// TIA Portal V20 export
DATA_BLOCK "Config"   // DB142
// stored: MemoryReserve 100, Namespace Unit1.Em0
   VAR
      em : "LAF_typeEmConfiguration";   // Configuration of EM Parameters
      cmStacker1NgBoxDetect : "LBC_typeDigitalSignalConfiguration";
      cmStacker1NgBoxFullDetect : "LBC_typeDigitalSignalConfiguration";
      cmStacker1NgBoxLoadingUpDown : "LBC_typeTwoWayActuatorConfiguration";
      cmStacker1NgBoxUnitMoverBwdFwd : "LBC_typeTwoWayActuatorConfiguration";
      cmStacker1NgBoxClampLeftOpenClose : "LBC_typeTwoWayActuatorConfiguration";
      cmStacker1NgBoxClampRightOpenClose : "LBC_typeTwoWayActuatorConfiguration";
      cmStacker1NgBoxClampMoverOpenClose : "LBC_typeTwoWayActuatorConfiguration";
      cmStacker1NgBoxLiftDownUp : "LBC_typeTwoWayActuatorConfiguration";
      cmStacker1NgBoxLockDownUp : "LBC_typeTwoWayActuatorConfiguration";
   END_VAR
BEGIN
   em.referenceDesignator.parent := WSTRING#'U1';
   em.referenceDesignator.relative := WSTRING#'EM0';
   cmStacker1NgBoxLoadingUpDown.referenceDesignator := WSTRING#'STACK NG CLAMP Z-AXIS';
   cmStacker1NgBoxLoadingUpDown.monitoringDiscrepancy := T#5s;
   cmStacker1NgBoxUnitMoverBwdFwd.referenceDesignator := WSTRING#'NG CLAMP UNIT MOVER';
   cmStacker1NgBoxUnitMoverBwdFwd.monitoringLeavingFeedback := T#10s;
   cmStacker1NgBoxUnitMoverBwdFwd.monitoringReachingFeedback := T#10s;
   cmStacker1NgBoxUnitMoverBwdFwd.monitoringDiscrepancy := T#5s;
   cmStacker1NgBoxClampLeftOpenClose.referenceDesignator := WSTRING#'STACK NG CLAMP LEFT';
   cmStacker1NgBoxClampLeftOpenClose.monitoringDiscrepancy := T#5s;
   cmStacker1NgBoxClampRightOpenClose.referenceDesignator := WSTRING#'STACK NG CLAMP RIGHT';
   cmStacker1NgBoxClampRightOpenClose.monitoringDiscrepancy := T#5s;
   cmStacker1NgBoxClampMoverOpenClose.referenceDesignator := WSTRING#'STACK NG CLAMP MOVER';
   cmStacker1NgBoxClampMoverOpenClose.monitoringDiscrepancy := T#5s;
   cmStacker1NgBoxLiftDownUp.referenceDesignator := WSTRING#'STACK NG BOX LIFT';
   cmStacker1NgBoxLiftDownUp.monitoringDiscrepancy := T#5s;
   cmStacker1NgBoxLockDownUp.referenceDesignator := WSTRING#'STACK NG BOX LOCK';
   cmStacker1NgBoxLockDownUp.monitoringReachingFeedback := T#5s;
   cmStacker1NgBoxLockDownUp.monitoringDiscrepancy := T#5s;
END_DATA_BLOCK
